// TwinCAT 3 PLC project MAS516
// ProgramVersion: 3.1.4026.13
// libraries:
//   CmpBitmapPool, * (System)
//   Tc2_Standard, * (Beckhoff Automation GmbH)
//   Tc2_System, * (Beckhoff Automation GmbH)
//   Tc3_Module, * (Beckhoff Automation GmbH)
//   VisuDialogs, * (System)
//   VisuSymbols,3.5.10.0,System
// project tree:
//   DUTs/ E_Status.TcDUT (not stored)
//   Enums/ E_CTRL_SIGNAL_TYPE.TcDUT (not stored)
//   Function Blocks/ DisplacementSumWithFiller.TcPOU (not stored), FB_AnalogInputScaling.TcPOU (not stored), FB_Clock.TcPOU (not stored), FB_ClosedLoopControlPID_DC.TcPOU (not stored), FB_ClosedLoopControl_PID.TcPOU (not stored), FB_DisplacementControl.TcPOU (not stored), FB_Encoder.TcPOU (not stored), FB_Integrator.TcPOU (not stored), FB_Joystick.TcPOU (not stored), FB_JoystickInputScaling.TcPOU, FB_DisplacementValveOutput.TcPOU (not stored), FB_LogicBox2SC.TcPOU, FB_LogicBoxSC.TcPOU (not stored), FB_SineMotionGenerator.TcPOU (not stored), FB_StartPos.TcPOU (not stored), FB_ThDisplacement.TcPOU, FB_TRYClosedLoopControl_PID.TcPOU (not stored), FB_YokeInputScaling.TcPOU (not stored), FB_ValveOutput.TcPOU (not stored), F_Sine.TcPOU (not stored)
//   / GlobalTextList.TcGTLO (not stored), PlcTask.TcTTO (not stored), Visualization Manager.TcVMO (not stored), VISU_TASK.TcTTO (not stored)
//   GVLs/ G_IO.TcGVL (not stored), G_Parameters.TcGVL (not stored), G_Sensors.TcGVL (not stored), HMI.TcGVL (not stored)
//   PID/ FB_ClosedLoopControl.TcPOU (not stored), FB_ClosedLoopControl_WODDY.TcPOU (not stored), PID_FBD.TcPOU (not stored)
//   POUs/ MAIN.TcPOU, P_HMI.TcPOU, P_Inputs.TcPOU (not stored), P_MotionControl.TcPOU, P_Outputs.TcPOU (not stored)
//   Struct/ ST_AnalogInputScaling.TcDUT (not stored), ST_JoystickInputScaling.TcDUT (not stored), ST_Platform.TcDUT (not stored), ST_YokeInputScaling.TcDUT (not stored), ST_Parameters.TcDUT (not stored), ST_ValveDeadBand.TcDUT (not stored), ST_ValveOutput.TcDUT (not stored)
//   VISUs/ Header.TcVIS (not stored), ImagePool.TcIPO (not stored), Main_screen.TcVIS, Screen_PID_Control.TcVIS (not stored), Settings.TcVIS (not stored), TogelSwich.TcVIS (not stored), Visualization.TcVIS (not stored)

// ---- Function Blocks/FB_JoystickInputScaling.TcPOU
FUNCTION_BLOCK FB_JoystickInputScaling
VAR_INPUT
	bEnable 				: BOOL;
	nRawInput 				: INT;
	stJoystickInputScaling  : ST_JoystickInputScaling;
END_VAR
VAR_OUTPUT
	fNormalizedOutput 		: LREAL;
END_VAR
VAR
	fRawInput 				: LREAL;
	fTempInput 				: LREAL;
	fTempOutput 			: LREAL;
END_VAR

fRawInput := INT_TO_LREAL(nRawInput);

fTempInput := fRawInput - stJoystickInputScaling.fNeutralInputValue;

IF fTempInput > stJoystickInputScaling.fNeutralDeadband THEN
	fTempOutput := fTempInput/(stJoystickInputScaling.fMaxInputValue - stJoystickInputScaling.fNeutralInputValue);
ELSIF fTempInput < -stJoystickInputScaling.fNeutralDeadband THEN	
	fTempOutput := fTempInput/(stJoystickInputScaling.fNeutralInputValue - stJoystickInputScaling.fMinInputValue);
ELSE
	fTempOutput := 0.0;
END_IF

IF NOT(bEnable) THEN
	fNormalizedOutput := 0.0;
ELSE
	fNormalizedOutput := LIMIT(stJoystickInputScaling.fMinOutputValue, fTempOutput, stJoystickInputScaling.fMaxOutputValue);
END_IF

END_FUNCTION_BLOCK

// ---- Function Blocks/FB_LogicBox2SC.TcPOU
FUNCTION_BLOCK FB_LogicBox2SC
VAR_INPUT
	fSeconderyPIDOut: LREAL;
	P_OutputsbEnableWinch: BOOL;
	fWinchVelRefManualSC: LREAL;
END_VAR
VAR_OUTPUT
	fOutputSecondaryControl: LREAL;
END_VAR
VAR
	rtb_k1: LREAL;
	rtb_Lifting: LREAL;
END_VAR


(* Outputs for Atomic SubSystem: '<Root>/FB_LogicBox2SC' *)
(* MATLAB Function: '<S1>/ControlerLogicBlock1' *)
(* MATLAB Function 'FB_LogicBox2SC/ControlerLogicBlock1': '<S2>:1' *)
(* '<S2>:1:2' if VelrefJoy >= 0.0 *)

IF fWinchVelRefManualSC >= 0.0 THEN 
    (* '<S2>:1:3' k1 = 0.5; *)
    rtb_k1 := 0.5;
ELSE 
    (* '<S2>:1:4' else *)
    (* '<S2>:1:5' k1 = 0.25; *)
    rtb_k1 := 0.25;
END_IF;

(* End of MATLAB Function: '<S1>/ControlerLogicBlock1' *)


(* Sum: '<S1>/Sum' *)
rtb_k1 := fSeconderyPIDOut + rtb_k1;
(* Saturate: '<S1>/MidFilter' *)

IF rtb_k1 > 0.45 THEN 
    fOutputSecondaryControl := 0.45;
ELSIF rtb_k1 >= 0.4 THEN 
    fOutputSecondaryControl := rtb_k1;
ELSE 
    fOutputSecondaryControl := 0.4;
END_IF;

(* End of Saturate: '<S1>/MidFilter' *)


(* Saturate: '<S1>/Lifting' *)

IF rtb_k1 > 0.65 THEN 
    rtb_Lifting := 0.65;
ELSIF rtb_k1 >= 0.5 THEN 
    rtb_Lifting := rtb_k1;
ELSE 
    rtb_Lifting := 0.5;
END_IF;

(* End of Saturate: '<S1>/Lifting' *)


(* Saturate: '<S1>/Lowring' *)

IF rtb_k1 > 0.30 THEN 
    rtb_k1 := 0.30;
ELSIF rtb_k1 < 0.12 THEN 
    rtb_k1 := 0.12;
END_IF;

(* End of Saturate: '<S1>/Lowring' *)


(* MATLAB Function: '<S1>/ControlerLogicBlock2' *)
(* Check if the input u is positive *)
(* MATLAB Function 'FB_LogicBox2SC/ControlerLogicBlock2': '<S3>:1' *)
(* '<S3>:1:3' if u > 0.0 *)

IF fWinchVelRefManualSC > 0.0 THEN 
    (* '<S3>:1:4' y = umax; *)
    fOutputSecondaryControl := rtb_Lifting;
    (* Output is 0.5 + u, capped at 0.6 for positive input *)
ELSIF fWinchVelRefManualSC < 0.0 THEN 
    (* '<S3>:1:5' elseif u < 0.0 *)
    (* '<S3>:1:6' y = umin; *)
    fOutputSecondaryControl := rtb_k1;
    (* Output is 0.25 + u, not dropping below 0.15 for negative input *)
END_IF;

(* End of MATLAB Function: '<S1>/ControlerLogicBlock2' *)


(* Switch: '<S1>/Switch1' *)

IF  NOT P_OutputsbEnableWinch THEN 
    (* Outport: '<Root>/fOutputSecondaryControl' incorporates:
     *  Constant: '<S1>/Constant1' *)
    fOutputSecondaryControl := 0.4;
END_IF;

(* End of Switch: '<S1>/Switch1' *)
(* End of Outputs for SubSystem: '<Root>/FB_LogicBox2SC' *)

END_FUNCTION_BLOCK

// ---- Function Blocks/FB_ThDisplacement.TcPOU
FUNCTION_BLOCK FB_ThDisplacement
VAR_INPUT
	stParam : ST_Parameters; 
	fDeltaP : LREAL;
END_VAR
VAR_OUTPUT
	fDisplacement : LREAL;
END_VAR
VAR
	fGravity : LREAL := 9.81; 
END_VAR

fDisplacement := (fGravity*stParam.fPayloadMass)/LIMIT(0.000001, fDeltaP*1E5, 400.0*1E5);

END_FUNCTION_BLOCK

// ---- POUs/MAIN.TcPOU
PROGRAM MAIN
VAR
	bStatusOk : BOOL;
	bFault : BOOL := FALSE;
	eStatus : E_Status := E_Status.Checking;
	bRunning : BOOL := TRUE;
	fCycleTime : LREAL:= 0.001;
	fTime : LREAL:= 0.0;
	fbPID_FBD : PID_FBD;
	Clock : FB_Clock; 
	bTest : BOOL;
	fTest : LREAL;
	
END_VAR

P_Inputs();
P_Outputs();
P_MotionControl();
P_HMI();
	
F_Sine(fTime:= fTime, SinuSignal=>G_IO.SinuSignal);
fbPID_FBD(ssMethodType :=1, In1:= G_IO.PositionError , Out1=> G_IO.PIDout); 

IF G_IO.bEmgOk AND NOT(G_IO.bStopButton) AND NOT(G_IO.bOffSwtich) AND NOT(bFault) THEN
	bStatusOk := TRUE;
ELSE 
	bStatusOk := FALSE;
END_IF

CASE eStatus OF 
	E_Status.Checking:
		IF bFault THEN
			eStatus := E_Status.Fault;
		END_IF
		
		IF bStatusOk THEN	
			eStatus := E_Status.Ready;
		END_IF
		
		IF NOT(bStatusOk) THEN	
			eStatus := E_Status.Off;
		END_IF
		
	E_Status.Off:	
		IF bStatusOk THEN	
			eStatus := E_Status.Checking;
		END_IF
		
		IF bFault THEN
			eStatus := E_Status.Fault;
		END_IF

	E_Status.Fault:
		IF NOT(bFault) THEN
			eStatus := E_Status.Checking;
		END_IF
	
	E_Status.Ready:
		IF G_IO.bStartButton AND bStatusOk AND NOT(bFault) THEN
			eStatus := E_Status.Starting;
		END_IF	
		
		IF  NOT(bStatusOk) OR bFault THEN
			eStatus := E_Status.Checking;
		END_IF	

	E_Status.Starting:
		IF bRunning THEN
			eStatus := E_Status.Running;
		END_IF 
		
		IF bFault OR NOT(bStatusOk)  THEN
			eStatus := E_Status.Checking;
		END_IF
		
	
	E_Status.Running:
	
		IF G_IO.bStopButton THEN
			eStatus := E_Status.Stopping;
		END_IF
		
		IF NOT(bRunning) OR NOT(bStatusOk) OR bFault THEN
			eStatus := E_Status.Checking;
		END_IF
	
	E_Status.Stopping:	
		IF NOT(bRunning) THEN
			eStatus := E_Status.Checking;
		END_IF
	
		IF NOT(bStatusOk) OR bFault THEN
		eStatus := E_Status.Checking;
		END_IF	
	
ELSE 	
	eStatus := E_Status.Checking;
END_CASE

END_PROGRAM

// ---- POUs/P_MotionControl.TcPOU
PROGRAM P_MotionControl
VAR
	fbClock : FB_Clock;
	fTime : LREAL;
	bStartClock : BOOL;
	fbPrimaryControl : FB_ClosedLoopControl; 
	fPGain : LREAL := G_IO.P_Gain;//3.0;
	fIGain : LREAL := G_IO.I_Gain;//1.0;
	fbJoystick : FB_Joystick;
	fWinchVelRef : LREAL;
	fWinchPosRef : LREAL;
	fbWinchVelIntegrator : FB_Integrator;
	fbEncoder : FB_Encoder;
	fWinchPos : LREAL;
	fInitialWinchPos : LREAL;
	bWinchVelIntegratorOn: BOOL := TRUE; 
	fSineMotionGen : FB_SineMotionGenerator;
	PosRefTEST : LREAL; 
	bAutoEnable : BOOL;
	bManualEnable : BOOL;
	fSineDisplacementSp : LREAL := 0.3; // Nils Was here
	fSinePeriodeTime : LREAL := 5.0;
	fWinchPosRefManual : LREAL;
	// fWinchPosRefAuto : LREAL;  // THis is in the G_IO.fWinchPosRefAuto for HMI
	fbGetStartPos : FB_StartPos;
	fWinchVelRefManual : LREAL;
	fWinchVelRefAuto : LREAL;
	
	// Primary Control
	fWinchControlOutput : LREAL;
	fOutputPrimaryControl : LREAL;
	fInputSecondaryControl : LREAL := 1.0; 
	
	// Secoder control 
	fbSecondaryControl: FB_ClosedLoopControl;
	fOutputSecondaryControl : LREAL := 1.0;
	fSecondaryControlPGain : LREAL := 3.0; 
	fSecondaryControlIGain : LREAL := 1.0; 
	
 
	
	//Displacement Control
	fDisplacementNormalizedInput : LREAL := 1.0;
	fDisplacementInitial : LREAL := 1.0;
	fbDisplacementControl : FB_ClosedLoopControl;
	fDisplacementControlSignal : LREAL;
	fMaxDisplacement : LREAL := 1.0;
	fMinDisplacement : LREAL := 0.0;
	fbThDisplacement : FB_ThDisplacement;
	fThDisplacement_m3 : LREAL;
	fThDisplacement_cm3 : LREAL;
	fThDisplacement_norm : LREAL;
	
	/// Nils Was Here
	fDisplacementControldTryRef : LREAL; 
	fDisplacementControldLowring: LREAL; 
	fDisplacementControldHoysting: LREAL;
		
 	fDisplacementControldMinum: LREAL;
	fGOODHELPSIN : FB_SineMotionGenerator; 
	fSineDisplacementTest: LREAL; 
	fbTickTock : FB_Clock;
	 
	fSumControlerWithFilter : DisplacementSumWithFiller;
	
	
	fSeconderyPIDOut : LREAL; 
	
	//fWinchPosRefManualSC: LREAL;
	//fWinchVelRefManualSC: LREAL;   
	
	fbWinchVelIntegratorSC : FB_Integrator; 
	fbLogicBoxSC : FB_LogicBoxSC;
	
	fVelRefCos : LREAL; 
	ftestPostionrefSC: LREAL; 
	
	fbClosedLoopControlDC   : FB_ClosedLoopControlPID_DC; 
	fDisplacementControlPgainDC : LREAL := 2.0;
	fDisplacementControlIgainDC : LREAL := 2.0;
	fDisplacementControlDgainDC : LREAL := 2.0;
	fDerativeFilterCoeffientDC 	: LREAL := 100; 
 
	IntgrtorON : BOOL; 
	
	DomLineTest : LREAL; 
	fTestSignal : LREAL;
	fbLogicBoxSCz : FB_LogicBox2SC; 
	fTimeSC : LREAL; 
	
	fWinchPosRefSC : LREAL;
	
END_VAR
VAR // added by the converter: edge detectors and wires of the graphical bodies
    _w1 : INT;
    _w2, _w3 : BOOL;
END_VAR

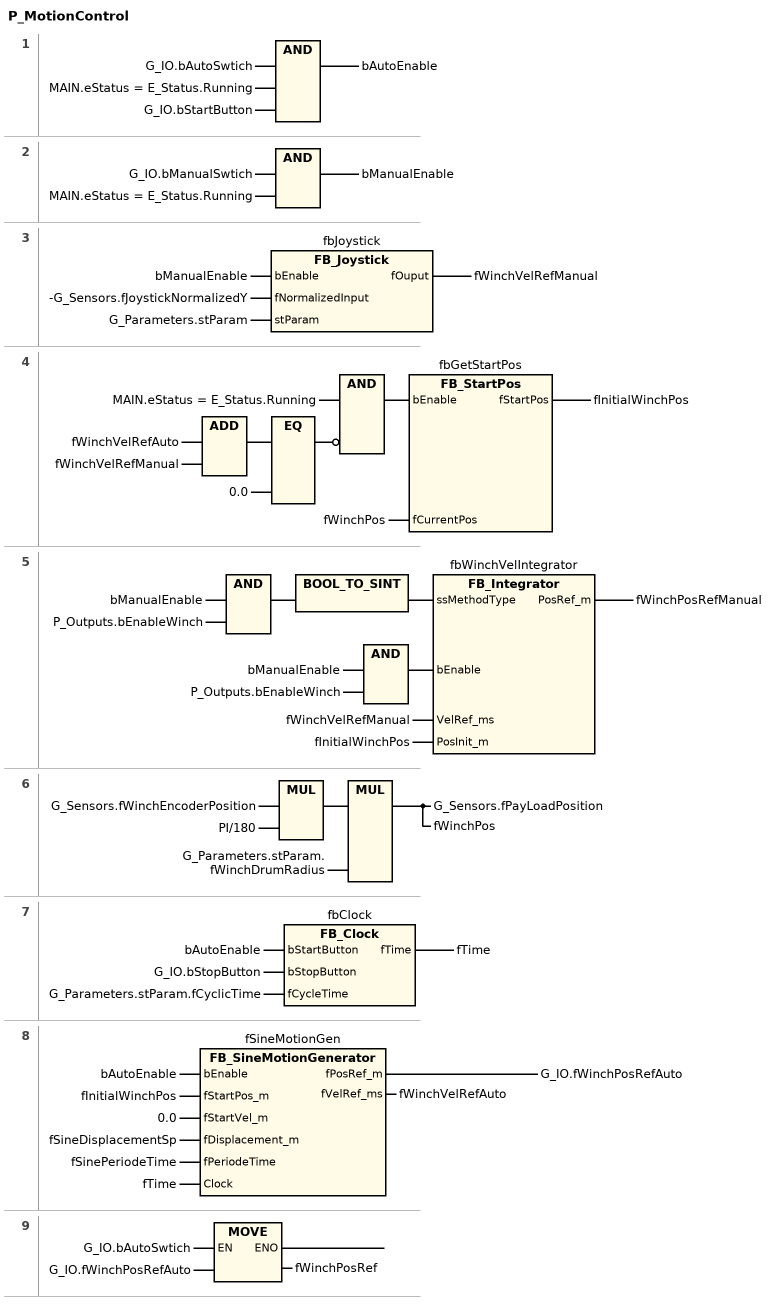
// NETWORK 1
bAutoEnable := G_IO.bAutoSwtich AND (MAIN.eStatus = E_Status.Running) AND G_IO.bStartButton;

// NETWORK 2
bManualEnable := G_IO.bManualSwtich AND (MAIN.eStatus = E_Status.Running);

// NETWORK 3
fbJoystick(
    bEnable := bManualEnable,
    fNormalizedInput := -G_Sensors.fJoystickNormalizedY,
    stParam := G_Parameters.stParam); // FB_Joystick
fWinchVelRefManual := fbJoystick.fOuput;

// NETWORK 4
fbGetStartPos(bEnable := (MAIN.eStatus = E_Status.Running) AND NOT (fWinchVelRefAuto + fWinchVelRefManual = 0.0), fCurrentPos := fWinchPos); // FB_StartPos
fInitialWinchPos := fbGetStartPos.fStartPos;

// NETWORK 5
fbWinchVelIntegrator(
    ssMethodType := BOOL_TO_SINT(bManualEnable AND P_Outputs.bEnableWinch),
    bEnable := bManualEnable AND P_Outputs.bEnableWinch,
    VelRef_ms := fWinchVelRefManual,
    PosInit_m := fInitialWinchPos); // FB_Integrator
fWinchPosRefManual := fbWinchVelIntegrator.PosRef_m;

// NETWORK 6
_w1 := (G_Sensors.fWinchEncoderPosition * (PI/180)) * G_Parameters.stParam.fWinchDrumRadius;
G_Sensors.fPayLoadPosition := _w1;
fWinchPos := _w1;

// NETWORK 7
fbClock(
    bStartButton := bAutoEnable,
    bStopButton := G_IO.bStopButton,
    fCycleTime := G_Parameters.stParam.fCyclicTime); // FB_Clock
fTime := fbClock.fTime;

// NETWORK 8
fSineMotionGen(
    bEnable := bAutoEnable,
    fStartPos_m := fInitialWinchPos,
    fStartVel_m := 0.0,
    fDisplacement_m := fSineDisplacementSp,
    fPeriodeTime := fSinePeriodeTime,
    Clock := fTime,
    fVelRef_ms => fWinchVelRefAuto); // FB_SineMotionGenerator
G_IO.fWinchPosRefAuto := fSineMotionGen.fPosRef_m;

// NETWORK 9
IF G_IO.bAutoSwtich THEN fWinchPosRef := G_IO.fWinchPosRefAuto; END_IF

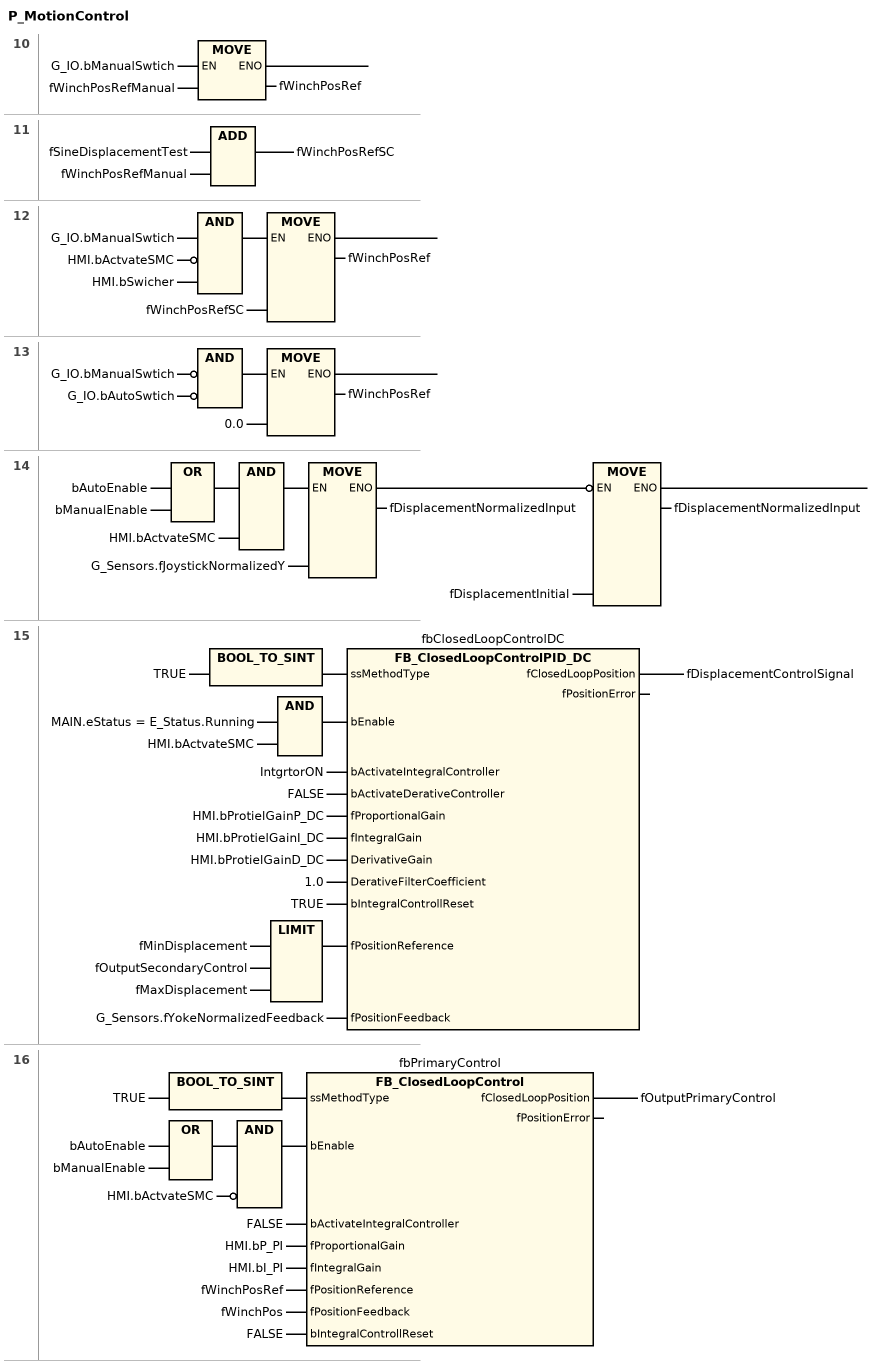
// NETWORK 10
IF G_IO.bManualSwtich THEN fWinchPosRef := fWinchPosRefManual; END_IF

// NETWORK 11
fWinchPosRefSC := fSineDisplacementTest + fWinchPosRefManual;

// NETWORK 12
IF G_IO.bManualSwtich AND NOT HMI.bActvateSMC AND HMI.bSwicher THEN fWinchPosRef := fWinchPosRefSC; END_IF

// NETWORK 13
IF NOT G_IO.bManualSwtich AND NOT G_IO.bAutoSwtich THEN fWinchPosRef := 0.0; END_IF

// NETWORK 14
_w2 := (bAutoEnable OR bManualEnable) AND HMI.bActvateSMC;
IF _w2 THEN fDisplacementNormalizedInput := G_Sensors.fJoystickNormalizedY; END_IF
IF NOT _w2 THEN fDisplacementNormalizedInput := fDisplacementInitial; END_IF

// NETWORK 15
fbClosedLoopControlDC(
    ssMethodType := BOOL_TO_SINT(TRUE),
    bEnable := (MAIN.eStatus = E_Status.Running) AND HMI.bActvateSMC,
    bActivateIntegralController := IntgrtorON,
    bActivateDerativeController := FALSE,
    fProportionalGain := HMI.bProtielGainP_DC,
    fIntegralGain := HMI.bProtielGainI_DC,
    DerivativeGain := HMI.bProtielGainD_DC,
    DerativeFilterCoefficient := 1.0,
    bIntegralControllReset := TRUE,
    fPositionReference := LIMIT(fMinDisplacement, fOutputSecondaryControl, fMaxDisplacement),
    fPositionFeedback := G_Sensors.fYokeNormalizedFeedback); // FB_ClosedLoopControlPID_DC
fDisplacementControlSignal := fbClosedLoopControlDC.fClosedLoopPosition;

// NETWORK 16
fbPrimaryControl(
    ssMethodType := BOOL_TO_SINT(TRUE),
    bEnable := (bAutoEnable OR bManualEnable) AND NOT HMI.bActvateSMC,
    bActivateIntegralController := FALSE,
    fProportionalGain := HMI.bP_PI,
    fIntegralGain := HMI.bI_PI,
    fPositionReference := fWinchPosRef,
    fPositionFeedback := fWinchPos,
    bIntegralControllReset := FALSE); // FB_ClosedLoopControl
fOutputPrimaryControl := fbPrimaryControl.fClosedLoopPosition;

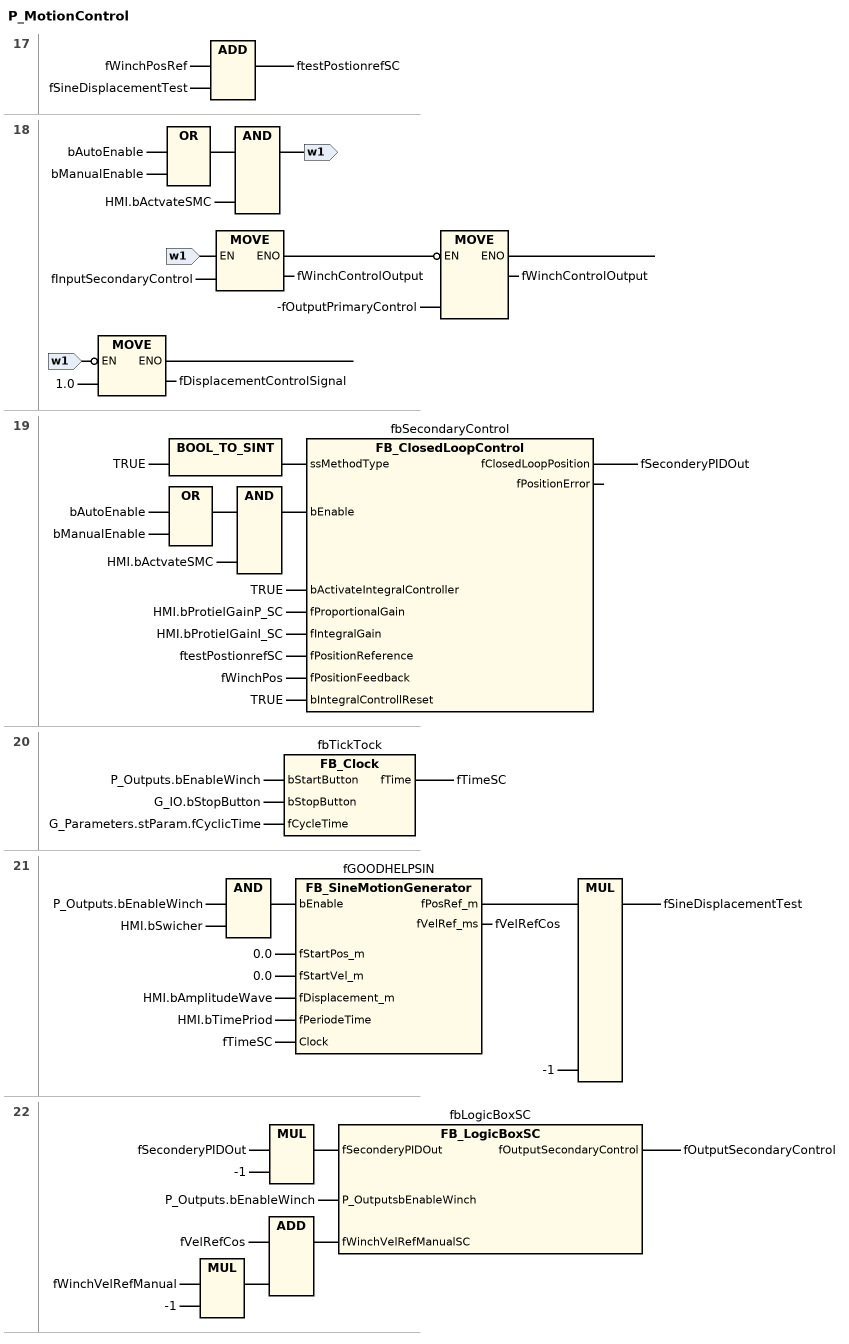
// NETWORK 17
ftestPostionrefSC := fWinchPosRef + fSineDisplacementTest;

// NETWORK 18
_w3 := (bAutoEnable OR bManualEnable) AND HMI.bActvateSMC;
IF _w3 THEN fWinchControlOutput := fInputSecondaryControl; END_IF
IF NOT _w3 THEN fWinchControlOutput := -fOutputPrimaryControl; END_IF
IF NOT _w3 THEN fDisplacementControlSignal := 1.0; END_IF

// NETWORK 19
fbSecondaryControl(
    ssMethodType := BOOL_TO_SINT(TRUE),
    bEnable := (bAutoEnable OR bManualEnable) AND HMI.bActvateSMC,
    bActivateIntegralController := TRUE,
    fProportionalGain := HMI.bProtielGainP_SC,
    fIntegralGain := HMI.bProtielGainI_SC,
    fPositionReference := ftestPostionrefSC,
    fPositionFeedback := fWinchPos,
    bIntegralControllReset := TRUE); // FB_ClosedLoopControl
fSeconderyPIDOut := fbSecondaryControl.fClosedLoopPosition;

// NETWORK 20
fbTickTock(
    bStartButton := P_Outputs.bEnableWinch,
    bStopButton := G_IO.bStopButton,
    fCycleTime := G_Parameters.stParam.fCyclicTime); // FB_Clock
fTimeSC := fbTickTock.fTime;

// NETWORK 21
fGOODHELPSIN(
    bEnable := P_Outputs.bEnableWinch AND HMI.bSwicher,
    fStartPos_m := 0.0,
    fStartVel_m := 0.0,
    fDisplacement_m := HMI.bAmplitudeWave,
    fPeriodeTime := HMI.bTimePriod,
    Clock := fTimeSC,
    fVelRef_ms => fVelRefCos); // FB_SineMotionGenerator
fSineDisplacementTest := fGOODHELPSIN.fPosRef_m * -1;

// NETWORK 22
fbLogicBoxSC(
    fSeconderyPIDOut := fSeconderyPIDOut * -1,
    P_OutputsbEnableWinch := P_Outputs.bEnableWinch,
    fWinchVelRefManualSC := fVelRefCos + fWinchVelRefManual * -1); // FB_LogicBoxSC
fOutputSecondaryControl := fbLogicBoxSC.fOutputSecondaryControl;

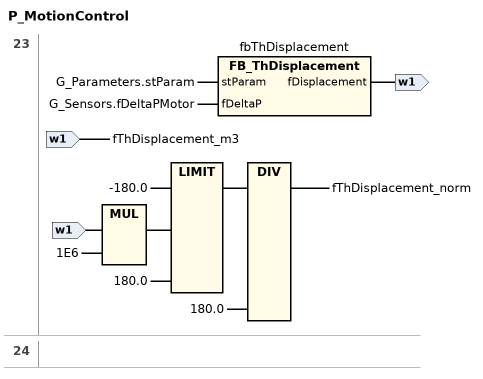
// NETWORK 23
fbThDisplacement(stParam := G_Parameters.stParam, fDeltaP := G_Sensors.fDeltaPMotor); // FB_ThDisplacement
fThDisplacement_m3 := fbThDisplacement.fDisplacement;
fThDisplacement_norm := LIMIT(-180.0, fbThDisplacement.fDisplacement * 1E6, 180.0) / 180.0;

// NETWORK 24

END_PROGRAM

// ---- POUs/P_HMI.TcPOU
PROGRAM P_HMI

VAR
    //bBlink : BOOL; // This variable toggles to create the blinking effect.
    tBlinkTimer : TON; // TON timer for controlling the blink rate.

	
	tSampleTimer: TON; // Timer for controlling the sampling rate
    nIndex: INT := 1; // Index for the next sample to be stored

END_VAR


HMI.bData1 := HMI.bP_PI; 
G_IO.P_Gain := HMI.bP_PI;

HMI.bDataP_DC := HMI.bProtielGainP_DC; 
HMI.bDataP_DC := HMI.bProtielGainP_DC; 


HMI.bData2 := HMI.bI_PI; 
G_IO.I_Gain := HMI.bI_PI;
// Enbiling the Ovrider fore END Stop //// 
/// HMI.bEndStopOverride := 

 

// Set the timer. It will start counting when IN is TRUE and reset when IN is FALSE.
tBlinkTimer(IN := NOT tBlinkTimer.Q, PT := T#1S); // The timer period is set to 1 second.

// Toggle the blink variable when the timer elapses (Q turns TRUE).
IF HMI.bEndStopOverride THEN
	IF tBlinkTimer.Q THEN
		HMI.bBlink := NOT HMI.bBlink;
	END_IF;
ELSE 
	HMI.bBlink := FALSE;
	
END_IF; 


IF HMI.bSwichForPlot THEN
	IF tBlinkTimer.Q THEN
		HMI.bSampleReady := NOT HMI.bSampleReady;
	END_IF;
ELSE 
	HMI.bSwichForPlot := FALSE;
	
END_IF; 


// for ploting the pistion of the system on vizualizer 
IF HMI.bSampleReady THEN
    HMI.arrPayLoadPositions[nIndex] := G_Sensors.fPayLoadPosition; // Store the current position
    
    nIndex := nIndex + 1; // Move to the next index
    IF nIndex > 100 THEN
        nIndex := 1; // Reset the index to create a circular buffer
    END_IF;
    
   HMI.bSampleReady := FALSE; // Reset the sample trigger
END_IF;


// for ploting the Sin Wave on vizualizer 
IF HMI.bSampleReady THEN
    HMI.arrSinPayLoadPositions[nIndex] := G_IO.SinuSignal; // Store the current position
    
    nIndex := nIndex + 1; // Move to the next index
    IF nIndex > 100 THEN
        nIndex := 1; // Reset the index to create a circular buffer
    END_IF;
    
   HMI.bSampleReady := FALSE; // Reset the sample trigger
END_IF;



IF HMI.bActvateSMC THEN
	IF tBlinkTimer.Q THEN
		HMI.bSampleReady := NOT HMI.bSampleReady;
	END_IF;
ELSE 
	HMI.bActvateSMC := FALSE;
	
END_IF; 


// for ploting the pistion of the system on vizualizer 
IF HMI.bSampleReady THEN
    HMI.arrPayLoadPositions[nIndex] := G_Sensors.fYokeNormalizedFeedback; // Store the current position
    
    nIndex := nIndex + 1; // Move to the next index
    IF nIndex > 100 THEN
        nIndex := 1; // Reset the index to create a circular buffer
    END_IF;
    
   HMI.bSampleReady := FALSE; // Reset the sample trigger
END_IF;

END_PROGRAM

// ---- VISUs/Main_screen.TcVIS
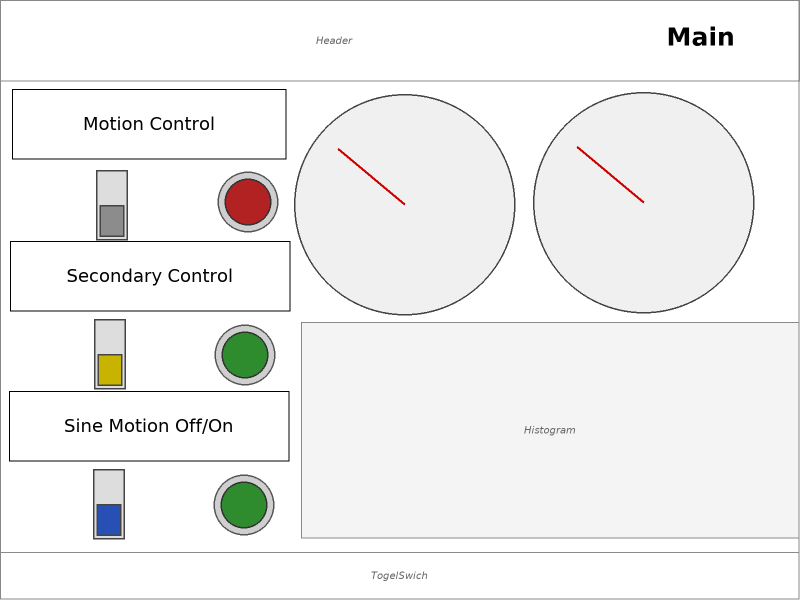
VISUALIZATION Main_screen  // 800x600
    Frame (-132,0 932x81)
        shows Header()
    Histogram (301,322 498x216), scale format: %.1f, scale 0..2
        p1518820177: G_Sensors.fPayLoadPosition
        p102497268: G_Sensors.fPayLoadPosition
    Meter360 (294,93 221x223), value: G_Sensors.fPressureWinchA, style: Meter-Meter360-Gray, scale format: %.1f, scale 0..100
        p518627256: PA bar
    Meter360 (533,91 221x223), value: G_Sensors.fPressureWinchB, style: Meter-Meter360-Gray, scale format: %.1f, scale 0..100
        p518627256: PB bar
    Frame (0,552 799x47)
        shows TogelSwich()
    Textfield (623,20 156x33), "Main"
    DipSwitch (30,319 160x70), variable: HMI.bActvateSMC, behaviour: TOGGLE, style: Switch-DipSwitch-Yellow
    Rectangle (10,241 280x70), "Secondary Control"
    Lamp1 (210,320 70x70), variable: not HMI.bActvateSMC, style: Lamp-Lamp1-Red
    Lamp1 (210,320 70x70), variable: HMI.bActvateSMC, invisible if: not HMI.bActvateSMC, style: Lamp-Lamp1-Green
    DipSwitch (29,469 160x70), variable: HMI.bSwicher, behaviour: TOGGLE, style: Switch-DipSwitch-Blue
    Rectangle (9,391 280x70), "Sine Motion Off/On"
    Lamp1 (209,470 70x70), variable: not HMI.bSwicher, style: Lamp-Lamp1-Red
    Lamp1 (209,470 70x70), variable: HMI.bSwicher, invisible if: not HMI.bSwicher, style: Lamp-Lamp1-Green
    Lamp1 (213,167 70x70), variable: HMI.bStartTB, invisible if: not HMI.bStartTB, style: Lamp-Lamp1-Green
    DipSwitch (32,170 160x70), variable: HMI.bStartTB, behaviour: TOGGLE, style: Switch-DipSwitch-Gray
    Rectangle (12,89 274x70), "Motion Control"
    Lamp1 (213,167 70x70), variable: not HMI.bStartTB, invisible if: HMI.bStartTB, style: Lamp-Lamp1-Red
END_VISUALIZATION
